// TIA Portal V18 export
VAR_GLOBAL   // PLC tag table "Run"
   Run_TF_Pump_Aeration_Clarifier_01 AT %Q3.5 : Bool;
   Run_TF_Pump_Aeration_Clarifier_02 AT %Q3.6 : Bool;
   Run_Suction_Pump_01 AT %Q0.6 : Bool;
   Run_Suction_Pump_02 AT %Q0.7 : Bool;
   Run_Suction_Pump_03 AT %Q1.0 : Bool;
   Run_Suction_Pump_04 AT %Q1.1 : Bool;
   Run_Suction_Pump_05 AT %Q1.2 : Bool;
   Run_Suction_Pump_06 AT %Q1.3 : Bool;
   Run_Suction_Pump_07 AT %Q1.4 : Bool;
   Run_Suction_Pump_08 AT %Q1.5 : Bool;
   Run_Backwash_Pump_01 AT %Q1.6 : Bool;
   Run_Backwash_Pump_02 AT %Q1.7 : Bool;
   Run_Backwash_Pump_03 AT %Q2.0 : Bool;
   Run_Backwash_Pump_04 AT %Q2.1 : Bool;
   Run_Backwash_Pump_05 AT %Q2.2 : Bool;
   Run_MBR_Aeration_01 AT %Q2.3 : Bool;
   Run_MBR_Aeration_02 AT %Q2.4 : Bool;
   Run_Chlorine_Dosing_Pump AT %Q2.5 : Bool;
   Run_Chlorine_Chemical_Agitator AT %Q2.6 : Bool;
   Run_Solid_TF_Clarifier AT %Q2.7 : Bool;
   Run_UV_1P_01 AT %Q3.0 : Bool;
   Run_UV_1P_02 AT %Q3.1 : Bool;
   Run_UV_1P_03 AT %Q3.2 : Bool;
   RUN_TF_PUMP_CSAS_B_01 AT %Q3.3 : Bool;
   RUN_TF_PUMP_CSAS_B_02 AT %Q3.4 : Bool;
   Run_TF_Pump_RWT_MMF_01 AT %Q3.7 : Bool;
   Run_TF_Pump_RWT_MMF_02 AT %Q4.0 : Bool;
   Run_PAC_Flocculant_Dosing_Pump AT %Q4.1 : Bool;
   Run_TF_Pump_Waterpool_Buffer_01 AT %Q4.2 : Bool;
   Run_TF_Pump_Waterpool_Buffer_02 AT %Q4.3 : Bool;
END_VAR
